TYPE ST_UserControl_Manual_Axis_Item :
STRUCT
	stName	: ST_Text;
	fPos	: LREAL;
END_STRUCT
END_TYPE

(* stored: Version 1.1.0.1, ProductVersion 3.1.4024.12
   DUT ST_UserControl_Manual_Axis_Item: Id {9f4b2d4b-2cda-443d-990b-e42d31c6fd30} *)
